(* CODESYS project Traffic_Light_1_RECOVERED.project

Project tree, tasks and I/O mapping:
  Device : CODESYS Control Win V3 x64, CODESYS, version 3.5.22.30
    application Application
      libraries: Standard, 3.5.22.0 (System)
      task VISU_TASK (cyclic, interval 100 ms, priority 31) calls VisuElems.Visu_Prg
      task MainTask (cyclic, interval t#20ms, priority 1) calls PLC_PRG
      visualisation Visualization
      program PLC_PRG [LD]
  text list GlobalTextList
*)

// Device/Application/PLC_PRG
PROGRAM PLC_PRG
VAR
	Stop: BOOL;
	Start: BOOL;
	Green: BOOL;
	Yellow: BOOL;
	Red: BOOL;
	TON_Green: TON;
	TON_Yellow: TON;
	TON_Red: TON;
	Run: BOOL;
	TON_RedQ: BOOL;
	TON_GreenQ: BOOL;
	TON_YellowQ: BOOL;
	Rec: BOOL;
	NO: BOOL;
	TON_Yellow1: TON;
	Ped_PB: BOOL;
	Ped_req: BOOL;
	TON_0: TON;
	TON_walk: TON;
	red_hold: BOOL;
END_VAR
VAR // added by the converter: edge detectors and wires of the graphical bodies
    _w1 : BOOL;
END_VAR

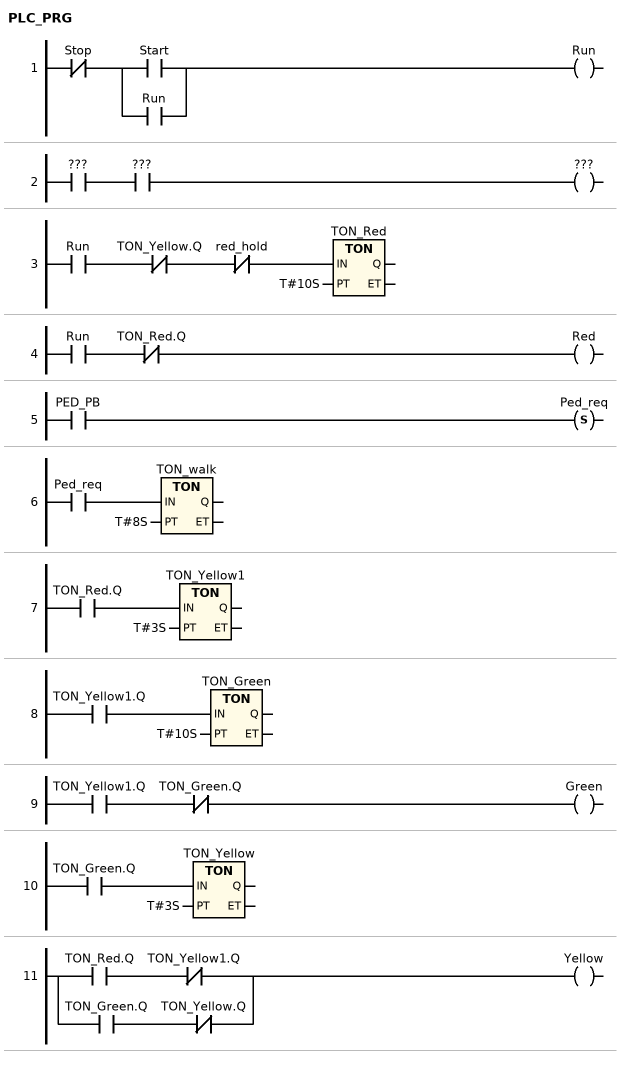
// NETWORK 1
_w1 := NOT Stop;
Run := _w1 AND Start OR _w1 AND Run;

// NETWORK 2
??? := ??? AND ???;

// NETWORK 3
TON_Red(IN := Run AND NOT TON_Yellow.Q AND NOT red_hold, PT := T#10S); // TON

// NETWORK 4
Red := Run AND NOT TON_Red.Q;

// NETWORK 5
Ped_req S= PED_PB;

// NETWORK 6
TON_walk(IN := Ped_req, PT := T#8S); // TON

// NETWORK 7
TON_Yellow1(IN := TON_Red.Q, PT := T#3S); // TON

// NETWORK 8
TON_Green(IN := TON_Yellow1.Q, PT := T#10S); // TON

// NETWORK 9
Green := TON_Yellow1.Q AND NOT TON_Green.Q;

// NETWORK 10
TON_Yellow(IN := TON_Green.Q, PT := T#3S); // TON

// NETWORK 11
Yellow := TON_Red.Q AND NOT TON_Yellow1.Q OR TON_Green.Q AND NOT TON_Yellow.Q;

END_PROGRAM

// Device/Application/Visualization
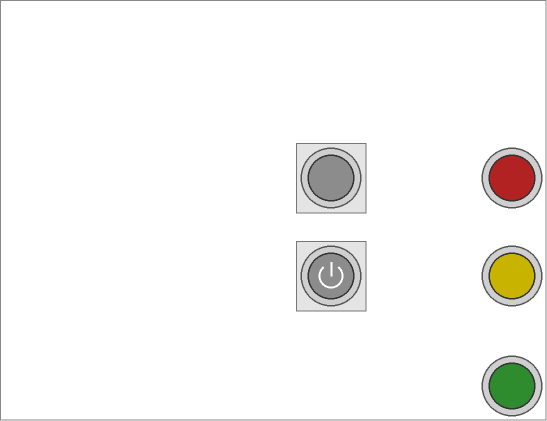
VISUALIZATION Visualization  // 547x421
    Lamp1 (477,143 70x70), variable: PLC_PRG.Red, style: Lamp-Lamp1-Red
    Lamp1 (477,241 70x70), variable: PLC_PRG.Yellow, style: Lamp-Lamp1-Yellow
    Lamp1 (477,351 70x70), variable: PLC_PRG.Green, style: Lamp-Lamp1-Green
    PowerSwitch (296,241 70x70), variable: PLC_PRG.Stop, behaviour: TOGGLE, style: Switch-PowerSwitch-Gray
    PushSwitch (296,143 70x70), variable: PLC_PRG.Start, behaviour: TOGGLE, style: Switch-PushSwitch-Gray
END_VISUALIZATION
